(* Schneider Machine Expert - Basic project ProyekAkhir_Muhammad Akmal Prabowo_2106708141, file version 2.7.0.0 *)
(* ProjectInformations: Name=New project *)

HARDWARE
  Cpu 0: TM221CE16R
  ModuleExtensionObject 0: TM2DDI32DK
  EthernetConfiguration: NetworkName=M221, IpAllocationMode=FixedAddress, IpAddress=0.0.0.0, SubnetMask=0.0.0.0
  SerialLineConfiguration: Baud=Baud19200, Parity=ParityEven, DataBits=DataBits8, StopBits=StopBits1, PhysicalMedium=PhysicalMediumRs485, TransmissionMode=TransmissionModeModbusRtu, SlaveId=1, Addressing=SlaveAddressing
  MastTask: UsePeriodScanMode=false, PeriodScan=100
  FastTask: Period=255
  CpuBehavior: StartingMode=StartAsPreviousState, AutoSaveRamOnEeprom=true, WatchdogPeriod=250

SYMBOLS  (address, symbol, comment, settings)
  %M0       STARTING  "Start"
  %M1       STOP  "Stop"
  %M2       EMERGENCY_STOP  "Emergency Stop"
  %M3       AUTO  "Auto"
  %M4       RESET  "Reset"
  %M5         "Diffuse sensor1"
  %M6       DIFFUSE_SENSOR_2  "Diffuse sensor2"
  %M7       BOX_AT_ENTRY  "RR sensor1"
  %M8       CLAMPED
  %M9         "plate _limit"
  %M10      PALLET_LOADED
  %M11      PALLET_AT_ENTRY
  %M16        "Conv main 1"
  %M17        "Conv main 2"
  %M18        "Conv med"
  %M19        "Conv high"
  %M20        "Pivot high"
  %M21        "Pivot belt high"
  %M22        "Pivot med"
  %M23        "Pivot belt med"
  %M50      START_CONV  "Start conv"
  %M51      MAIN_CONV  "Main conv"
  %M52      CONV_HIGH  "Conv high"
  %M53      CONV_MED  "Conv med"
  %M54      PIVOT_FOR_HIGH  "Pivot1"
  %M55      PIVOT_FOR_MED  "Pivot2"
  %M56      BELTPIVOT_FOR_HIGH  "Beltpivot1"
  %M57      BELTPIVOT_FOR_MED  "Beltpivot2"
  %M58      BOX_FEEDER  "Box feeder"
  %M59      LOAD_BELT  "Load belt"
  %M60      PUSH  "Palettizer pusher"
  %M61      OPEN_PLATE
  %M62      PALLET_FEEDER
  %M63      CLAMP
  %M64      LOAD_PALLET
  %M65      MOVE_TO_LIMIT
  %M66      ELEVATOR_UP
  %M67      ELEVATOR_DOWN
  %M68      EXIT_COVEYOR
  %M69      WARNING_LIGHT
  %TM0        [Preset=1, Base=OneSecond]
  %TM1        [Preset=3, Base=OneSecond]
  %TM2        [Preset=4, Base=OneSecond]
  %TM3        [Preset=2, Base=OneSecond]
  %TM4        [Preset=1, Base=OneSecond]
  %TM5        [Preset=3, Base=OneSecond]
  %TM6        [Preset=5, Base=OneSecond]
  %TM7        [Preset=6, Base=OneSecond]
  %TM8        [Preset=5, Base=OneSecond]
  %TM9        [Preset=55, Base=OneHundredMilliSeconds]
  %TM10       [Preset=3, Base=OneSecond]
  %TM11       [Preset=5, Base=OneSecond]
  %TM12       [Preset=2, Base=OneSecond]
  %I0.0       "Start button"
  %I0.1       "Stop button"

POU New POU
  (* SectionNumber=1 *)

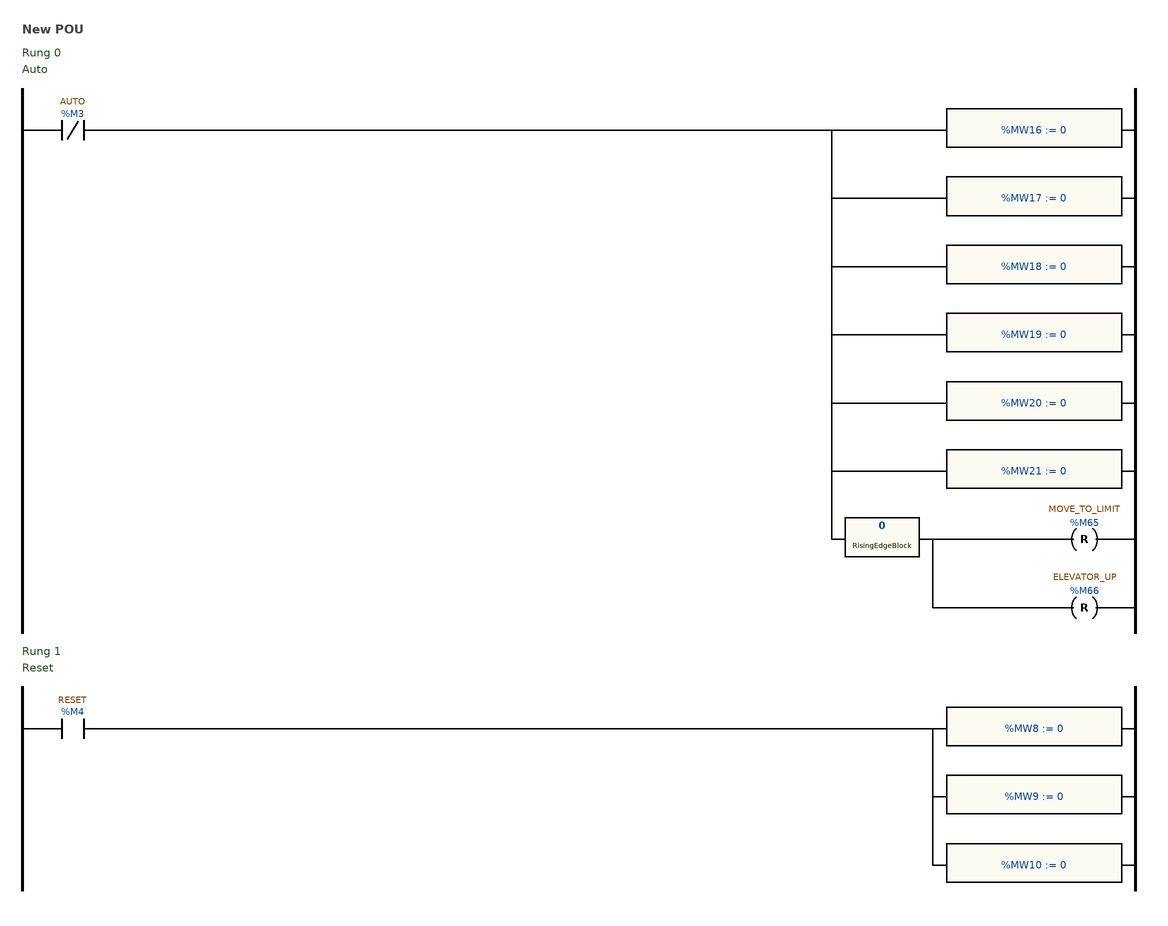

// Rung 0
// Auto
  LDN %M3                 (* AUTO *)
  MPS
  [ %MW16 := 0 ]
  MRD
  [ %MW17 := 0 ]
  MRD
  [ %MW18 := 0 ]
  MRD
  [ %MW19 := 0 ]
  MRD
  [ %MW20 := 0 ]
  MRD
  [ %MW21 := 0 ]
  MPP
  RISING0
  R %M65                  (* MOVE_TO_LIMIT *)
  R %M66                  (* ELEVATOR_UP *)
  // as ST:
  //   IF NOT AUTO THEN %MW16 := 0; END_IF;
  //   IF NOT AUTO THEN %MW17 := 0; END_IF;
  //   IF NOT AUTO THEN %MW18 := 0; END_IF;
  //   IF NOT AUTO THEN %MW19 := 0; END_IF;
  //   IF NOT AUTO THEN %MW20 := 0; END_IF;
  //   IF NOT AUTO THEN %MW21 := 0; END_IF;
  //   IF RISING(NOT AUTO) THEN MOVE_TO_LIMIT := FALSE; END_IF;
  //   IF RISING(NOT AUTO) THEN ELEVATOR_UP := FALSE; END_IF;

// Rung 1
// Reset
  LD %M4                  (* RESET *)
  [ %MW8 := 0 ]
  [ %MW9 := 0 ]
  [ %MW10 := 0 ]
  // as ST:
  //   IF RESET THEN %MW8 := 0; END_IF;
  //   IF RESET THEN %MW9 := 0; END_IF;
  //   IF RESET THEN %MW10 := 0; END_IF;

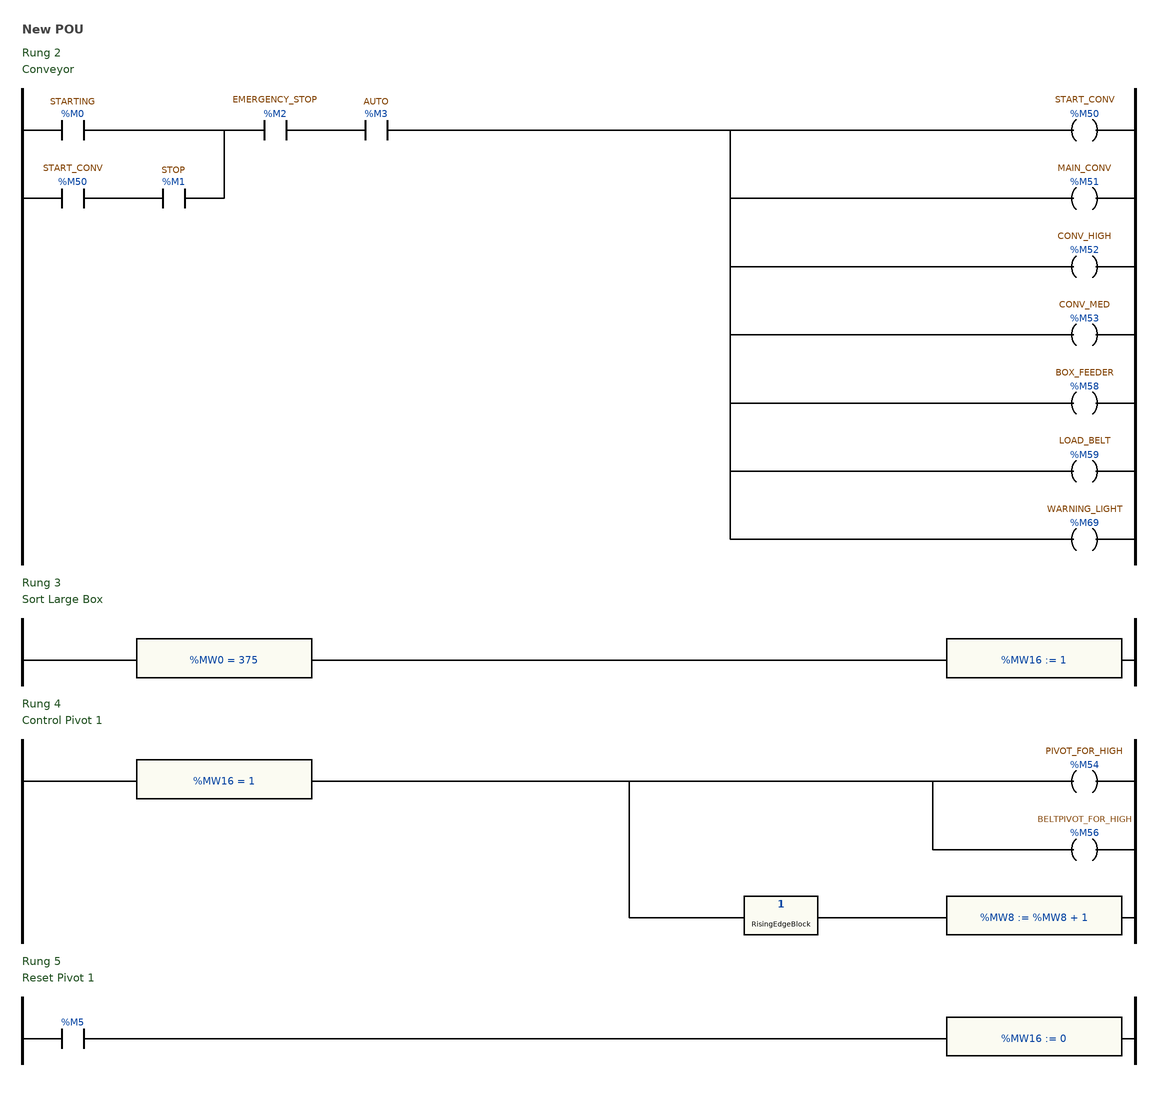

// Rung 2
// Conveyor
  LD %M0                  (* STARTING *)
  OR( %M50                (* START_CONV *)
  AND %M1                 (* STOP *)
  )
  AND %M2                 (* EMERGENCY_STOP *)
  AND %M3                 (* AUTO *)
  ST %M50                 (* START_CONV *)
  ST %M51                 (* MAIN_CONV *)
  ST %M52                 (* CONV_HIGH *)
  ST %M53                 (* CONV_MED *)
  ST %M58                 (* BOX_FEEDER *)
  ST %M59                 (* LOAD_BELT *)
  ST %M69                 (* WARNING_LIGHT *)
  // as ST:
  //   _t1 := (STARTING OR START_CONV AND STOP) AND EMERGENCY_STOP AND AUTO;
  //   START_CONV := _t1;
  //   MAIN_CONV := _t1;
  //   CONV_HIGH := _t1;
  //   CONV_MED := _t1;
  //   BOX_FEEDER := _t1;
  //   LOAD_BELT := _t1;
  //   WARNING_LIGHT := _t1;

// Rung 3
// Sort Large Box
  LD [ %MW0 = 375 ]
  [ %MW16 := 1 ]
  // as ST:
  //   IF %MW0 = 375 THEN %MW16 := 1; END_IF;

// Rung 4
// Control Pivot 1
  LD [ %MW16 = 1 ]
  MPS
  ST %M54                 (* PIVOT_FOR_HIGH *)
  ST %M56                 (* BELTPIVOT_FOR_HIGH *)
  MPP
  RISING1
  [ %MW8 := %MW8 + 1 ]
  // as ST:
  //   PIVOT_FOR_HIGH := %MW16 = 1;
  //   BELTPIVOT_FOR_HIGH := %MW16 = 1;
  //   IF RISING(%MW16 = 1) THEN %MW8 := %MW8 + 1; END_IF;

// Rung 5
// Reset Pivot 1
  LD %M5
  [ %MW16 := 0 ]
  // as ST:
  //   IF %M5 THEN %MW16 := 0; END_IF;

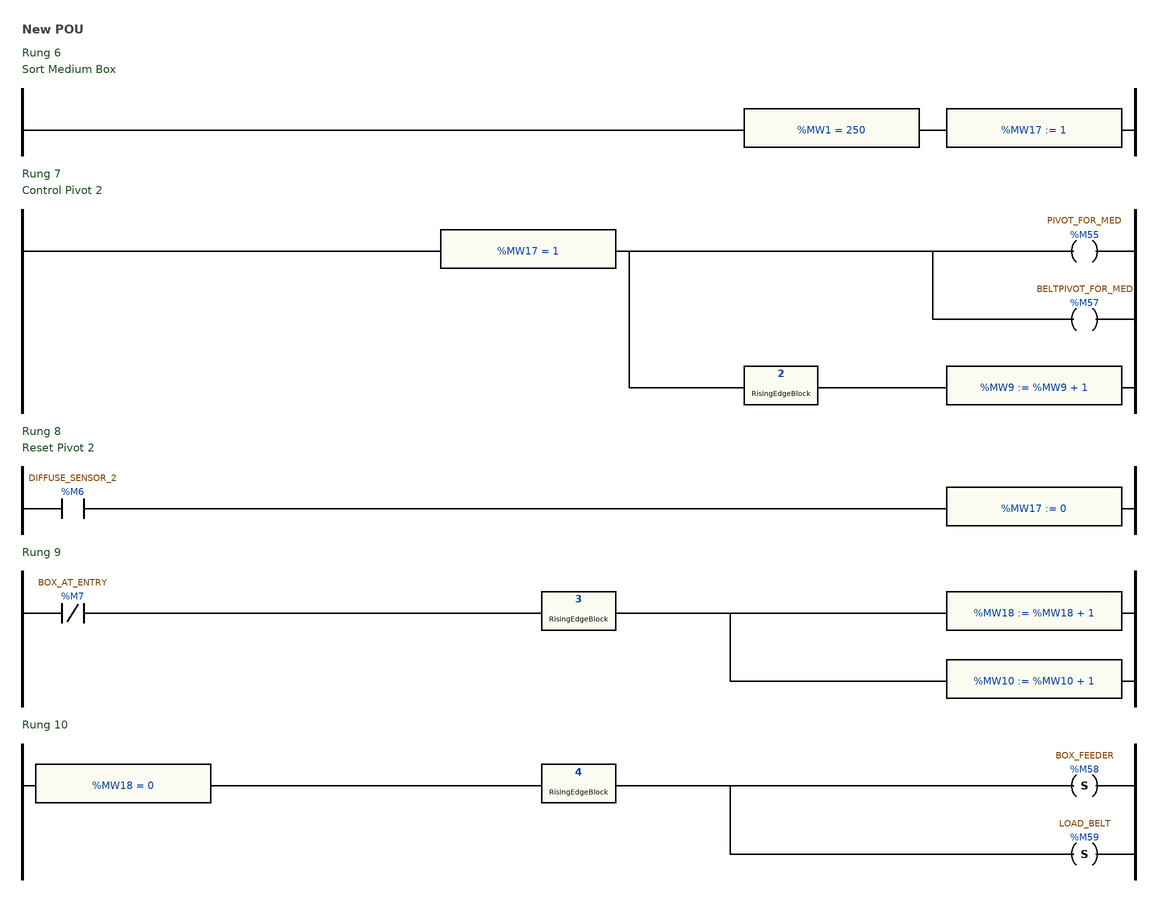

// Rung 6
// Sort Medium Box
  LD [ %MW1 = 250 ]
  [ %MW17 := 1 ]
  // as ST:
  //   IF %MW1 = 250 THEN %MW17 := 1; END_IF;

// Rung 7
// Control Pivot 2
  LD [ %MW17 = 1 ]
  MPS
  ST %M55                 (* PIVOT_FOR_MED *)
  ST %M57                 (* BELTPIVOT_FOR_MED *)
  MPP
  RISING2
  [ %MW9 := %MW9 + 1 ]
  // as ST:
  //   PIVOT_FOR_MED := %MW17 = 1;
  //   BELTPIVOT_FOR_MED := %MW17 = 1;
  //   IF RISING(%MW17 = 1) THEN %MW9 := %MW9 + 1; END_IF;

// Rung 8
// Reset Pivot 2
  LD %M6                  (* DIFFUSE_SENSOR_2 *)
  [ %MW17 := 0 ]
  // as ST:
  //   IF DIFFUSE_SENSOR_2 THEN %MW17 := 0; END_IF;

// Rung 9
  LDN %M7                 (* BOX_AT_ENTRY *)
  RISING3
  [ %MW18 := %MW18 + 1 ]
  [ %MW10 := %MW10 + 1 ]
  // as ST:
  //   IF RISING(NOT BOX_AT_ENTRY) THEN %MW18 := %MW18 + 1; END_IF;
  //   IF RISING(NOT BOX_AT_ENTRY) THEN %MW10 := %MW10 + 1; END_IF;

// Rung 10
  LD [ %MW18 = 0 ]
  RISING4
  S %M58                  (* BOX_FEEDER *)
  S %M59                  (* LOAD_BELT *)
  // as ST:
  //   IF RISING(%MW18 = 0) THEN BOX_FEEDER := TRUE; END_IF;
  //   IF RISING(%MW18 = 0) THEN LOAD_BELT := TRUE; END_IF;

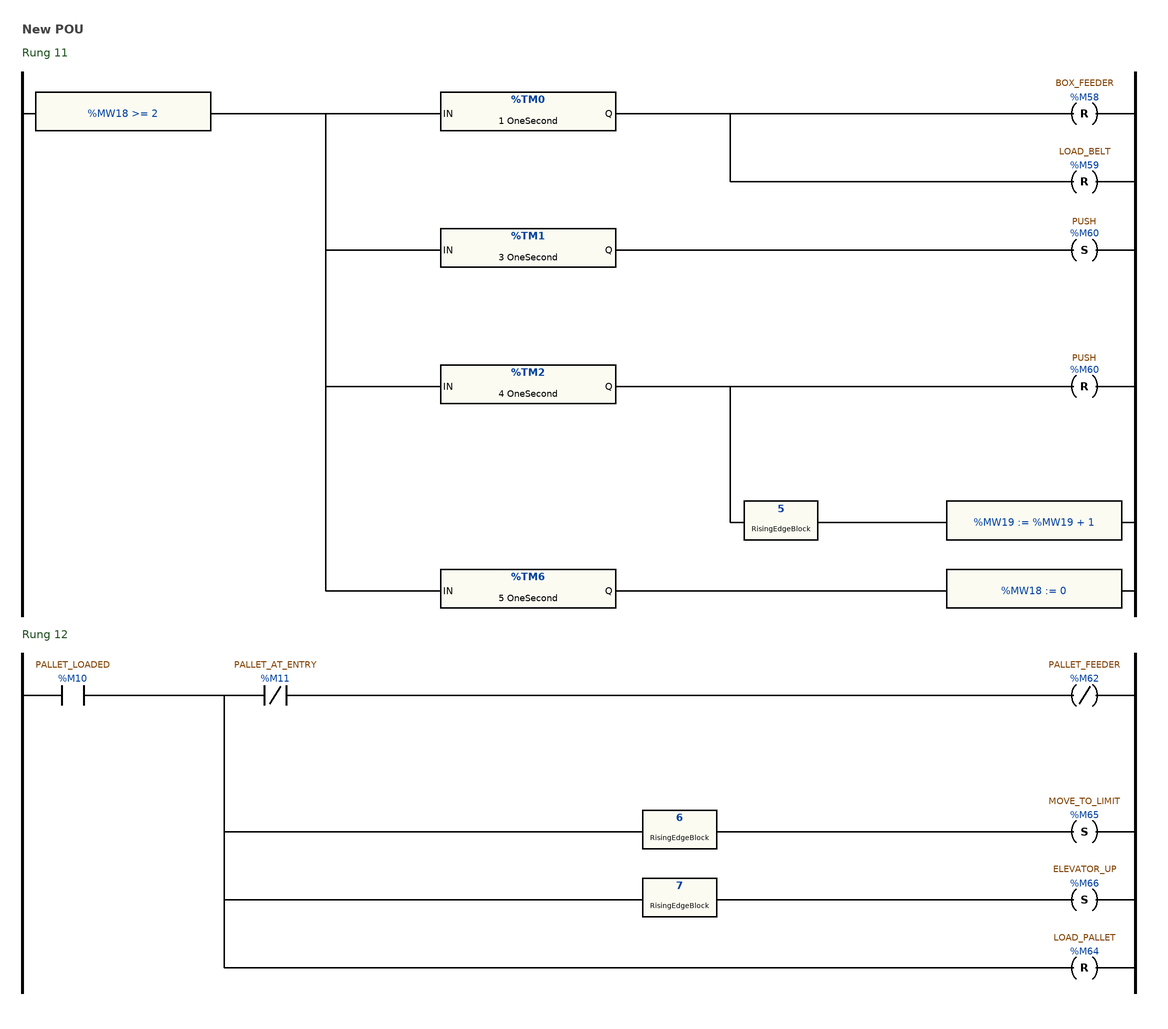

// Rung 11
  LD 1
  MULTIFB
  LD 1
  AND [ %MW18 >= 2 ]
  ST %MW2009:X0
  BLK %TM0
  LD %MW2009:X0
  IN
  OUT_BLK
  LD Q
  R %M58                  (* BOX_FEEDER *)
  R %M59                  (* LOAD_BELT *)
  END_BLK
  BLK %TM1
  LD %MW2009:X0
  IN
  OUT_BLK
  LD Q
  S %M60                  (* PUSH *)
  END_BLK
  BLK %TM2
  LD %MW2009:X0
  IN
  OUT_BLK
  LD Q
  MPS
  R %M60                  (* PUSH *)
  MPP
  RISING5
  [ %MW19 := %MW19 + 1 ]
  END_BLK
  BLK %TM6
  LD %MW2009:X0
  IN
  OUT_BLK
  LD Q
  [ %MW18 := 0 ]
  END_BLK
  MULTIFB
  // as ST:
  //   %TM0(IN := %MW18 >= 2);
  //   IF %TM0.Q THEN BOX_FEEDER := FALSE; END_IF;
  //   IF %TM0.Q THEN LOAD_BELT := FALSE; END_IF;
  //   %TM1(IN := %MW18 >= 2);
  //   IF %TM1.Q THEN PUSH := TRUE; END_IF;
  //   %TM2(IN := %MW18 >= 2);
  //   IF %TM2.Q THEN PUSH := FALSE; END_IF;
  //   IF RISING(%TM2.Q) THEN %MW19 := %MW19 + 1; END_IF;
  //   %TM6(IN := %MW18 >= 2);
  //   IF %TM6.Q THEN %MW18 := 0; END_IF;

// Rung 12
  LD %M10                 (* PALLET_LOADED *)
  MPS
  ANDN %M11               (* PALLET_AT_ENTRY *)
  STN %M62                (* PALLET_FEEDER *)
  MRD
  RISING6
  S %M65                  (* MOVE_TO_LIMIT *)
  MRD
  RISING7
  S %M66                  (* ELEVATOR_UP *)
  MPP
  R %M64                  (* LOAD_PALLET *)
  // as ST:
  //   PALLET_FEEDER := NOT (PALLET_LOADED AND NOT PALLET_AT_ENTRY);
  //   IF RISING(PALLET_LOADED) THEN MOVE_TO_LIMIT := TRUE; END_IF;
  //   IF RISING(PALLET_LOADED) THEN ELEVATOR_UP := TRUE; END_IF;
  //   IF PALLET_LOADED THEN LOAD_PALLET := FALSE; END_IF;

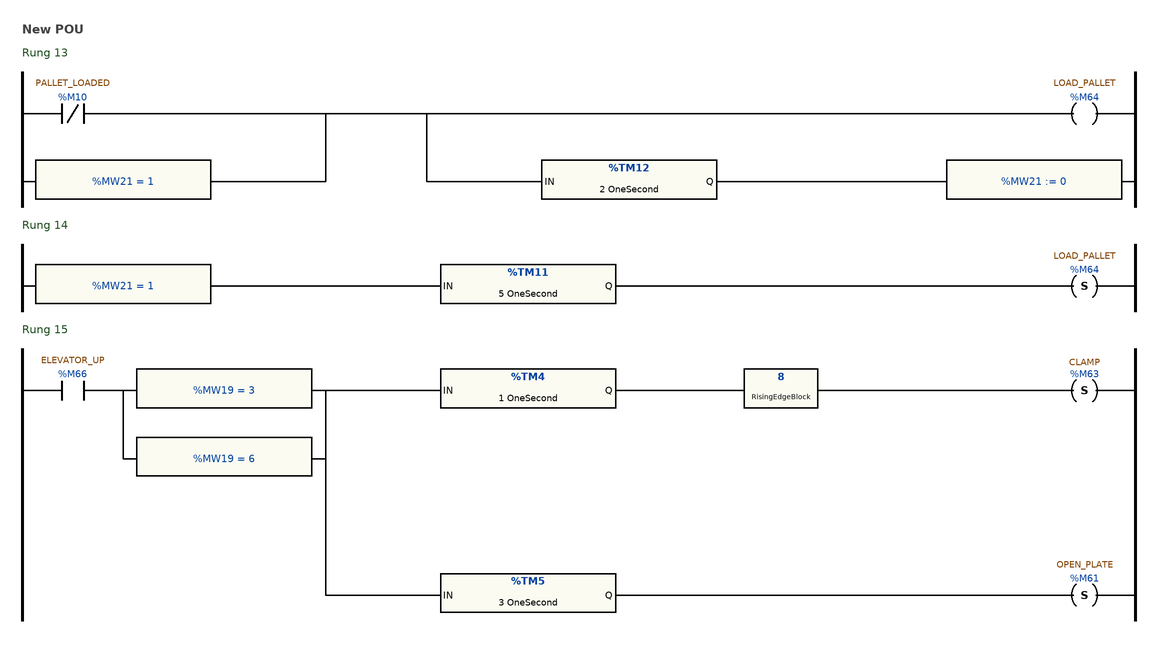

// Rung 13
  LD 1
  MULTIFB
  LD 1
  ANDN %M10               (* PALLET_LOADED *)
  OR [ %MW21 = 1 ]
  ST %MW2009:X0
  LD %MW2009:X0
  ST %M64                 (* LOAD_PALLET *)
  BLK %TM12
  LD %MW2009:X0
  IN
  OUT_BLK
  LD Q
  [ %MW21 := 0 ]
  END_BLK
  MULTIFB
  // as ST:
  //   LOAD_PALLET := NOT PALLET_LOADED OR %MW21 = 1;
  //   %TM12(IN := NOT PALLET_LOADED OR %MW21 = 1);
  //   IF %TM12.Q THEN %MW21 := 0; END_IF;

// Rung 14
  BLK %TM11
  LD [ %MW21 = 1 ]
  IN
  OUT_BLK
  LD Q
  S %M64                  (* LOAD_PALLET *)
  END_BLK
  // as ST:
  //   %TM11(IN := %MW21 = 1);
  //   IF %TM11.Q THEN LOAD_PALLET := TRUE; END_IF;

// Rung 15
  LD 1
  MULTIFB
  LD 1
  AND %M66                (* ELEVATOR_UP *)
  AND( [ %MW19 = 3 ]
  OR [ %MW19 = 6 ]
  )
  ST %MW2009:X0
  BLK %TM4
  LD %MW2009:X0
  IN
  OUT_BLK
  LD Q
  RISING8
  S %M63                  (* CLAMP *)
  END_BLK
  BLK %TM5
  LD %MW2009:X0
  IN
  OUT_BLK
  LD Q
  S %M61                  (* OPEN_PLATE *)
  END_BLK
  MULTIFB
  // as ST:
  //   %TM4(IN := ELEVATOR_UP AND (%MW19 = 3 OR %MW19 = 6));
  //   IF RISING(%TM4.Q) THEN CLAMP := TRUE; END_IF;
  //   %TM5(IN := ELEVATOR_UP AND (%MW19 = 3 OR %MW19 = 6));
  //   IF %TM5.Q THEN OPEN_PLATE := TRUE; END_IF;

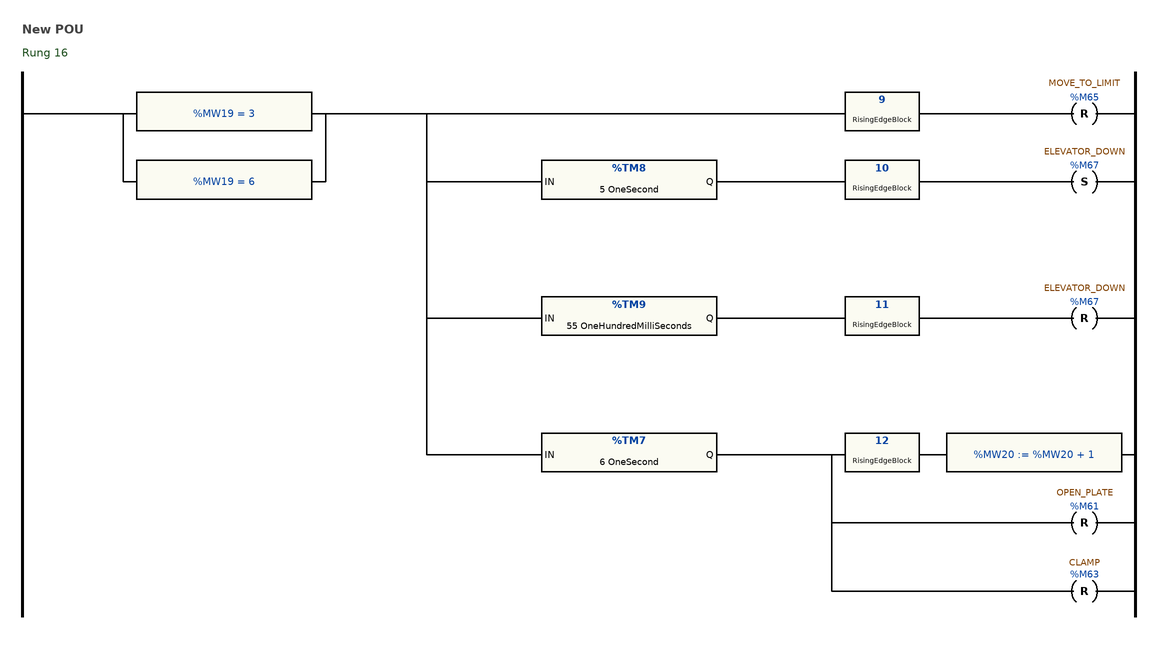

// Rung 16
  LD 1
  MULTIFB
  LD 1
  AND( [ %MW19 = 3 ]
  OR [ %MW19 = 6 ]
  )
  ST %MW2009:X0
  LD %MW2009:X0
  RISING9
  R %M65                  (* MOVE_TO_LIMIT *)
  BLK %TM8
  LD %MW2009:X0
  IN
  OUT_BLK
  LD Q
  RISING10
  S %M67                  (* ELEVATOR_DOWN *)
  END_BLK
  BLK %TM9
  LD %MW2009:X0
  IN
  OUT_BLK
  LD Q
  RISING11
  R %M67                  (* ELEVATOR_DOWN *)
  END_BLK
  BLK %TM7
  LD %MW2009:X0
  IN
  OUT_BLK
  LD Q
  MPS
  RISING12
  [ %MW20 := %MW20 + 1 ]
  MRD
  R %M61                  (* OPEN_PLATE *)
  MPP
  R %M63                  (* CLAMP *)
  END_BLK
  MULTIFB
  // as ST:
  //   IF RISING(%MW19 = 3 OR %MW19 = 6) THEN MOVE_TO_LIMIT := FALSE; END_IF;
  //   %TM8(IN := %MW19 = 3 OR %MW19 = 6);
  //   IF RISING(%TM8.Q) THEN ELEVATOR_DOWN := TRUE; END_IF;
  //   %TM9(IN := %MW19 = 3 OR %MW19 = 6);
  //   IF RISING(%TM9.Q) THEN ELEVATOR_DOWN := FALSE; END_IF;
  //   %TM7(IN := %MW19 = 3 OR %MW19 = 6);
  //   IF RISING(%TM7.Q) THEN %MW20 := %MW20 + 1; END_IF;
  //   IF %TM7.Q THEN OPEN_PLATE := FALSE; END_IF;
  //   IF %TM7.Q THEN CLAMP := FALSE; END_IF;

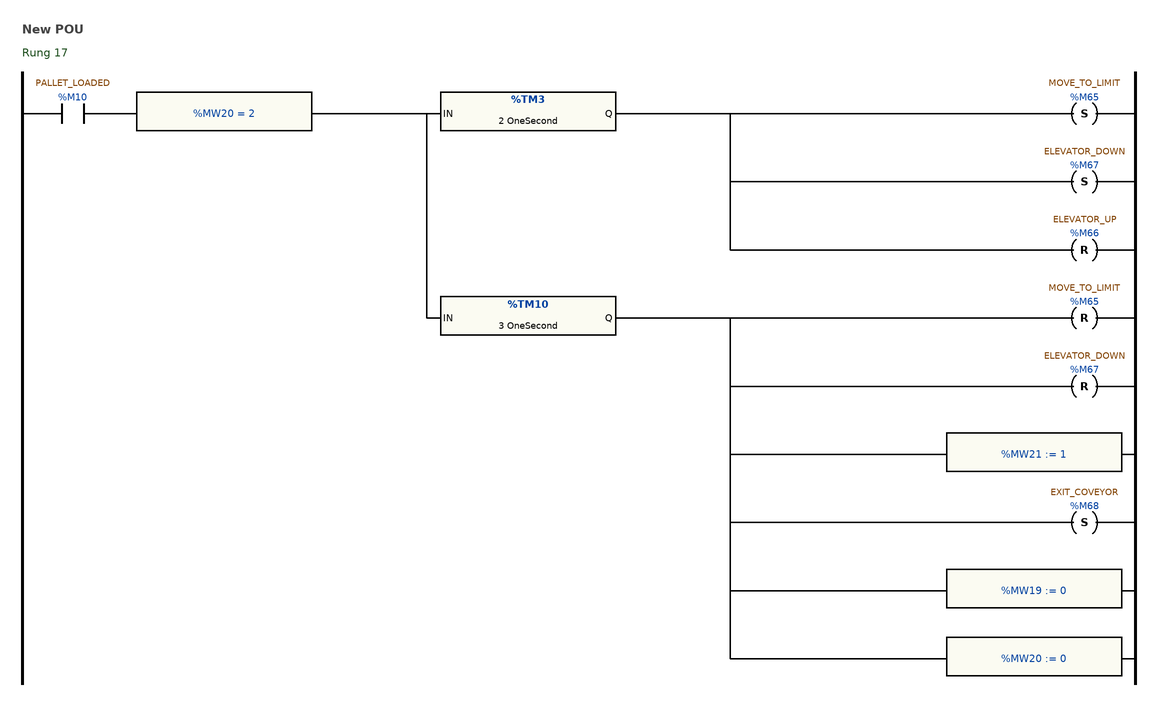

// Rung 17
  LD 1
  MULTIFB
  LD 1
  AND %M10                (* PALLET_LOADED *)
  AND [ %MW20 = 2 ]
  ST %MW2009:X0
  BLK %TM3
  LD %MW2009:X0
  IN
  OUT_BLK
  LD Q
  S %M65                  (* MOVE_TO_LIMIT *)
  S %M67                  (* ELEVATOR_DOWN *)
  R %M66                  (* ELEVATOR_UP *)
  END_BLK
  BLK %TM10
  LD %MW2009:X0
  IN
  OUT_BLK
  LD Q
  R %M65                  (* MOVE_TO_LIMIT *)
  R %M67                  (* ELEVATOR_DOWN *)
  [ %MW21 := 1 ]
  S %M68                  (* EXIT_COVEYOR *)
  [ %MW19 := 0 ]
  [ %MW20 := 0 ]
  END_BLK
  MULTIFB
  // as ST:
  //   %TM3(IN := PALLET_LOADED AND %MW20 = 2);
  //   IF %TM3.Q THEN MOVE_TO_LIMIT := TRUE; END_IF;
  //   IF %TM3.Q THEN ELEVATOR_DOWN := TRUE; END_IF;
  //   IF %TM3.Q THEN ELEVATOR_UP := FALSE; END_IF;
  //   %TM10(IN := PALLET_LOADED AND %MW20 = 2);
  //   IF %TM10.Q THEN MOVE_TO_LIMIT := FALSE; END_IF;
  //   IF %TM10.Q THEN ELEVATOR_DOWN := FALSE; END_IF;
  //   IF %TM10.Q THEN %MW21 := 1; END_IF;
  //   IF %TM10.Q THEN EXIT_COVEYOR := TRUE; END_IF;
  //   IF %TM10.Q THEN %MW19 := 0; END_IF;
  //   IF %TM10.Q THEN %MW20 := 0; END_IF;
